VAR_GLOBAL CONSTANT
	MAX_D_IN	: INT := 100;
END_VAR

(* stored: Version 1.1.0.1, ProductVersion 3.1.0.36
   GVL IO_DigiIn_Parameters: Id {67abd78c-e76e-4800-a1ed-c6e56f6fbbbc}, ParameterList True *)
